// Mitsubishi GX Works2 project: PLC_Group_08   PLC: FX3G

// global labels: Global1
VAR_GLOBAL
  switch7 AT X007 : BOOL;
  lamp7 AT Y007 : BOOL;
  berry_input AT D1100 : INT;
  lemon_input AT D1102 : INT;
  stabilizer_input AT D1104 : INT;
  gum_input AT D1106 : INT;
  berry_stock AT D1200 : INT;
  lemon_stock AT D1202 : INT;
  stabilizer_stock AT D1204 : INT;
  gum_stock AT D1206 : INT;
  M_start AT M0 : BOOL;
  cooling_berry AT D1300 : INT;
  cooling_lemon AT D1302 : INT;
  storage AT D1304 : INT;
  switch5 AT X005 : BOOL;
  analog_input1 AT D8280 : INT;
  switch1 AT X001 : BOOL;
  save_analog_input1 AT D8202 : INT;
END_VAR
VAR_GLOBAL CONSTANT
  K_5 : INT := 2000;
  K_6 : INT := 2400;
  K_10 : INT := 4000;
END_VAR
VAR_GLOBAL
  M_normal AT M1 : BOOL;
  M_pinuk AT M2 : BOOL;
END_VAR
VAR_GLOBAL CONSTANT
  K_7 : INT := 7;
  K_berry_normal : INT := 280;
  K_berry_pinuk : INT := 385;
  K_lemon_normal : INT := 455;
  K_lemon_pinuk : INT := 665;
  K_gum_normal : INT := 28;
  K_gum_pinuk : INT := 70;
  K_stabilizer_normal : INT := 105;
  K_stabilizer_pinuk : INT := 210;
END_VAR
VAR_GLOBAL
  M_yes_stock AT M3 : BOOL;
  M_exit AT M4 : BOOL;
  berry_to_subtract AT D1500 : INT;
  lemon_to_subtract AT D1502 : INT;
  stabilizer_to_subtract AT D1504 : INT;
  gum_to_subtract AT D1506 : INT;
  making_berry AT D1306 : INT;
  making_lemon AT D1308 : INT;
  M_check_stock AT M5 : BOOL;
  M_make_icecream AT M6 : BOOL;
END_VAR
VAR_GLOBAL CONSTANT
  K_berry_total_normal : INT := 350;
  K_berry_total_pinuk : INT := 560;
  K_lemon_total_normal : INT := 490;
  K_lemon_total_pinuk : INT := 700;
END_VAR
VAR_GLOBAL
  berry_total AT D1508 : INT;
  lemon_total AT D1510 : INT;
  making_icecream_timer_c AT TC0 : BOOL;
END_VAR
VAR_GLOBAL CONSTANT
  K_50 : INT := 50;
END_VAR
VAR_GLOBAL
  making_icecream_timer_s AT TS0 : BOOL;
  lamp0 AT Y000 : BOOL;
  M_empty AT M7 : BOOL;
  M_cool_icecream AT M8 : BOOL;
  switch2 AT X002 : BOOL;
  cooling_icecream_timer_c AT TC1 : BOOL;
  cooling_icecream_timer_s AT TS1 : BOOL;
END_VAR
VAR_GLOBAL CONSTANT
  K_80 : INT := 80;
END_VAR
VAR_GLOBAL
  lamp2 AT Y002 : BOOL;
  switch3 AT X003 : BOOL;
  M_mix_materials AT M9 : BOOL;
  M_make_icecream_timer AT M11 : BOOL;
  M_cool_icecream_timer AT M10 : BOOL;
  mixing_container AT D1310 : INT;
END_VAR
VAR_GLOBAL CONSTANT
  K_mixing_total_normal : INT := 868;
  K_mixing_total_pinuk : INT := 1330;
  K_3 : INT := 3;
END_VAR
VAR_GLOBAL
  mixing_total AT D1512 : INT;
  mixing_duration AT D1514 : INT;
  M_mix_materials_timer AT M12 : BOOL;
  mix_materials_timer_c AT TC2 : BOOL;
  mix_materials_timer_s AT TS2 : BOOL;
  M_lamps_helper AT M13 : BOOL;
  lamp_5_timer_c AT TC3 : BOOL;
  lamp_5_timer_s AT TS3 : BOOL;
  lamp5 AT Y005 : BOOL;
  lamp_6_timer_c AT TC4 : BOOL;
  lamp_6_timer_s AT TS4 : BOOL;
  lamp6 AT Y006 : BOOL;
END_VAR
VAR_GLOBAL CONSTANT
  K_30 : INT := 30;
  K_01 : INT := 40;
  K_0 : INT;
END_VAR
VAR_GLOBAL
  M_berry_stock_check AT M14 : BOOL;
  M_lemon_stock_check AT M15 : BOOL;
  M_stabilizer_stock_check AT M16 : BOOL;
  M_gum_stock_check AT M17 : BOOL;
  analog_output AT D8282 : INT;
END_VAR
VAR_GLOBAL CONSTANT
  K_10_timer : INT := 10;
END_VAR
VAR_GLOBAL
  M_cool_and_mix AT M18 : BOOL;
END_VAR

// task Task_01 (event TRUE, interval 0, priority 31): POU_01

PROGRAM POU_01
(* structured ladder/FBD written out as ST: instructions are called as NAME(EN, inputs, outputs); _pN, _eN, _tN stand for wires *)
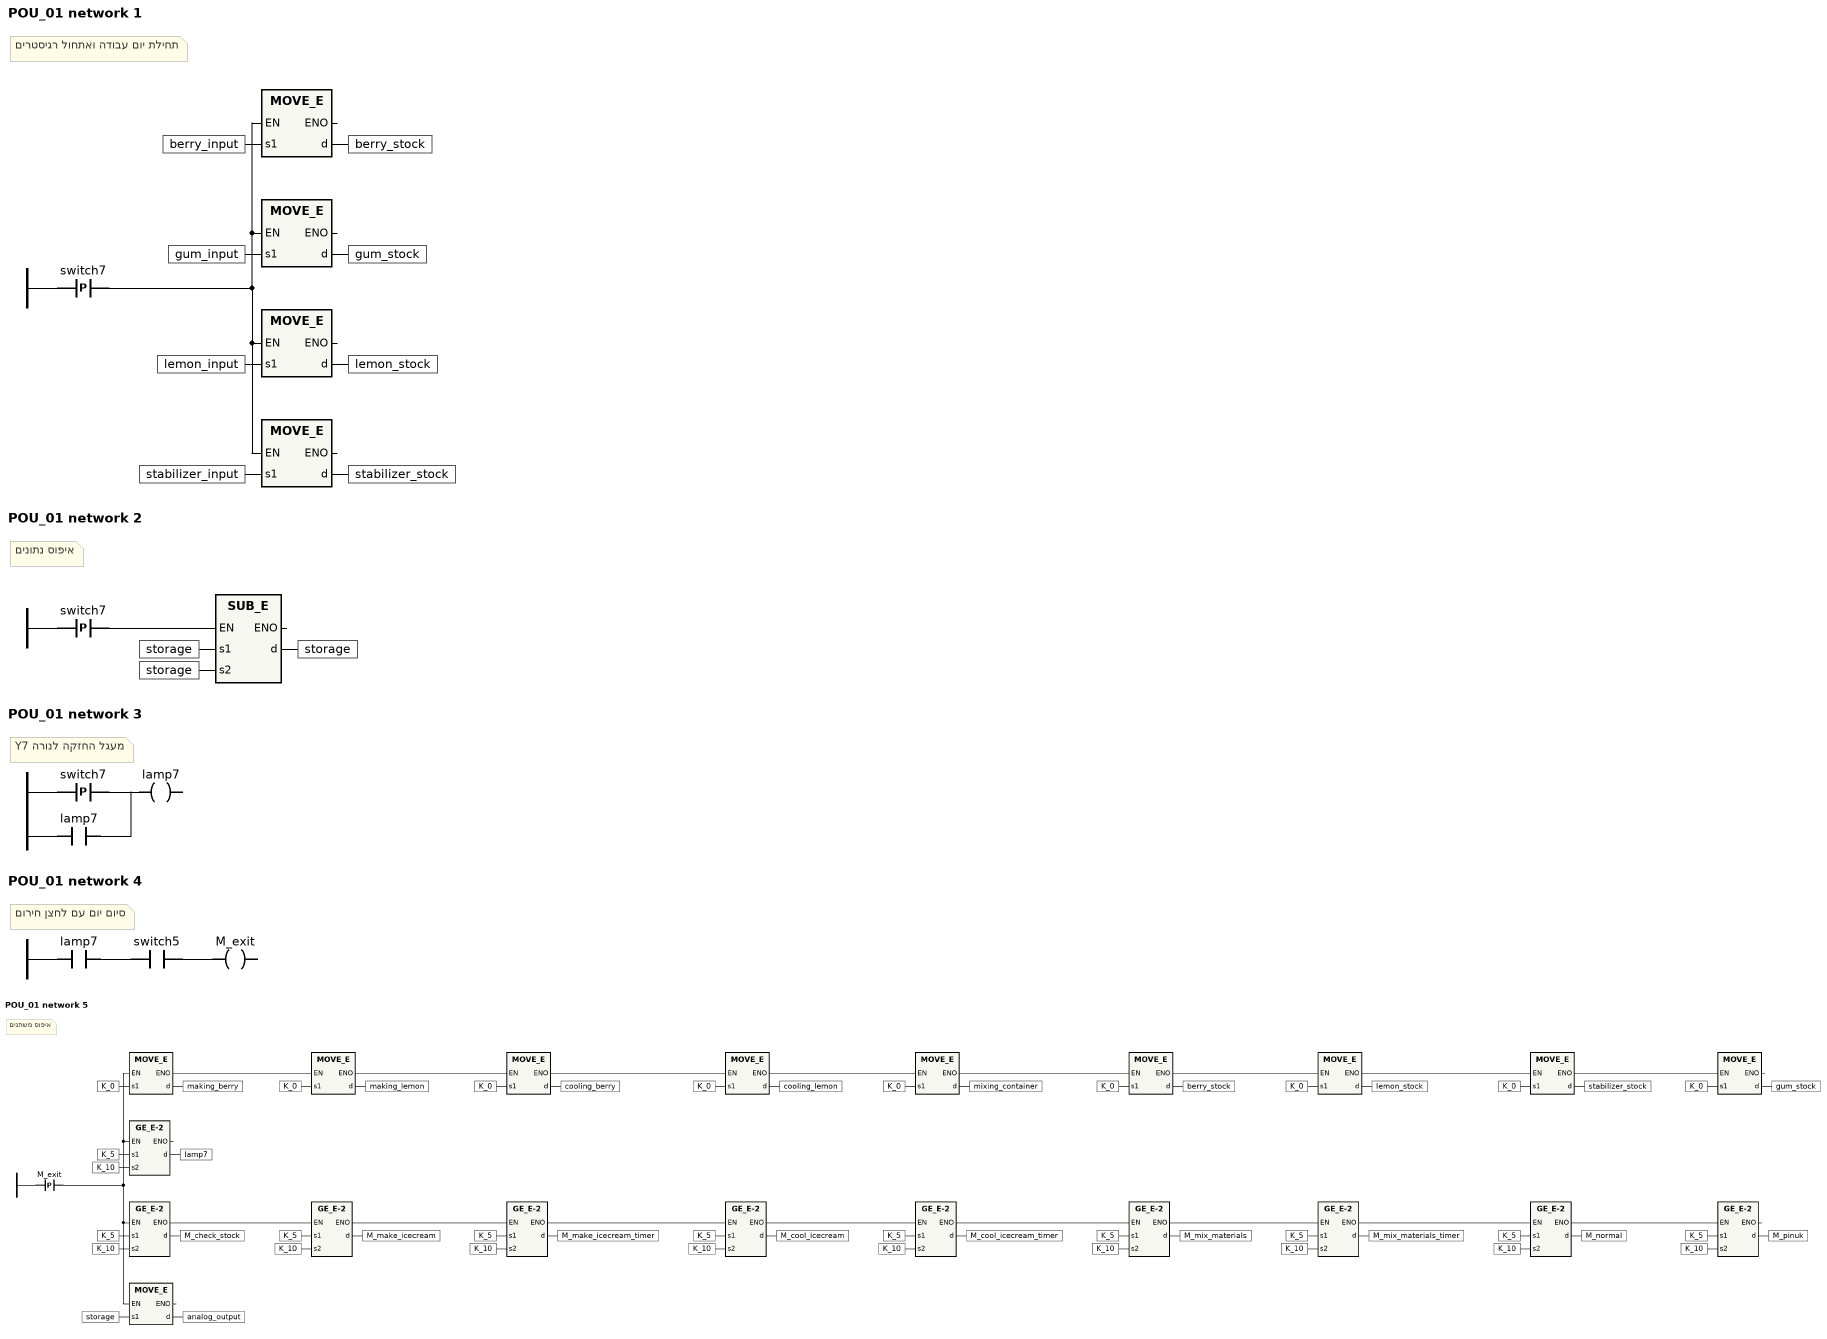
(* network 1 *)
(* תחילת יום עבודה ואתחול רגיסטרים *)
_p1 := LDP(TRUE, switch7);
MOVE_E(_p1, berry_input, berry_stock);
MOVE_E(_p1, gum_input, gum_stock);
MOVE_E(_p1, lemon_input, lemon_stock);
MOVE_E(_p1, stabilizer_input, stabilizer_stock);
(* network 2 *)
(* איפוס נתונים *)
SUB_E(LDP(TRUE, switch7), storage, storage, storage);
(* network 3 *)
(* מעגל החזקה לנורה Y7 *)
lamp7 := LDP(TRUE, switch7) OR lamp7;
(* network 4 *)
(* סיום יום עם לחצן חירום *)
M_exit := lamp7 AND switch5;
(* network 5 *)
(* איפוס משתנים *)
_p1 := LDP(TRUE, M_exit);
_e2 := MOVE_E(_p1, K_0, making_berry);
_e3 := MOVE_E(_e2, K_0, making_lemon);
_e4 := MOVE_E(_e3, K_0, cooling_berry);
_e5 := MOVE_E(_e4, K_0, cooling_lemon);
_e6 := MOVE_E(_e5, K_0, mixing_container);
_e7 := MOVE_E(_e6, K_0, berry_stock);
_e8 := MOVE_E(_e7, K_0, lemon_stock);
_e9 := MOVE_E(_e8, K_0, stabilizer_stock);
MOVE_E(_e9, K_0, gum_stock);
GE_E(_p1, K_5, K_10, lamp7);
_e10 := GE_E(_p1, K_5, K_10, M_check_stock);
_e11 := GE_E(_e10, K_5, K_10, M_make_icecream);
_e12 := GE_E(_e11, K_5, K_10, M_make_icecream_timer);
_e13 := GE_E(_e12, K_5, K_10, M_cool_icecream);
_e14 := GE_E(_e13, K_5, K_10, M_cool_icecream_timer);
_e15 := GE_E(_e14, K_5, K_10, M_mix_materials);
_e16 := GE_E(_e15, K_5, K_10, M_mix_materials_timer);
_e17 := GE_E(_e16, K_5, K_10, M_normal);
GE_E(_e17, K_5, K_10, M_pinuk);
MOVE_E(_p1, storage, analog_output);
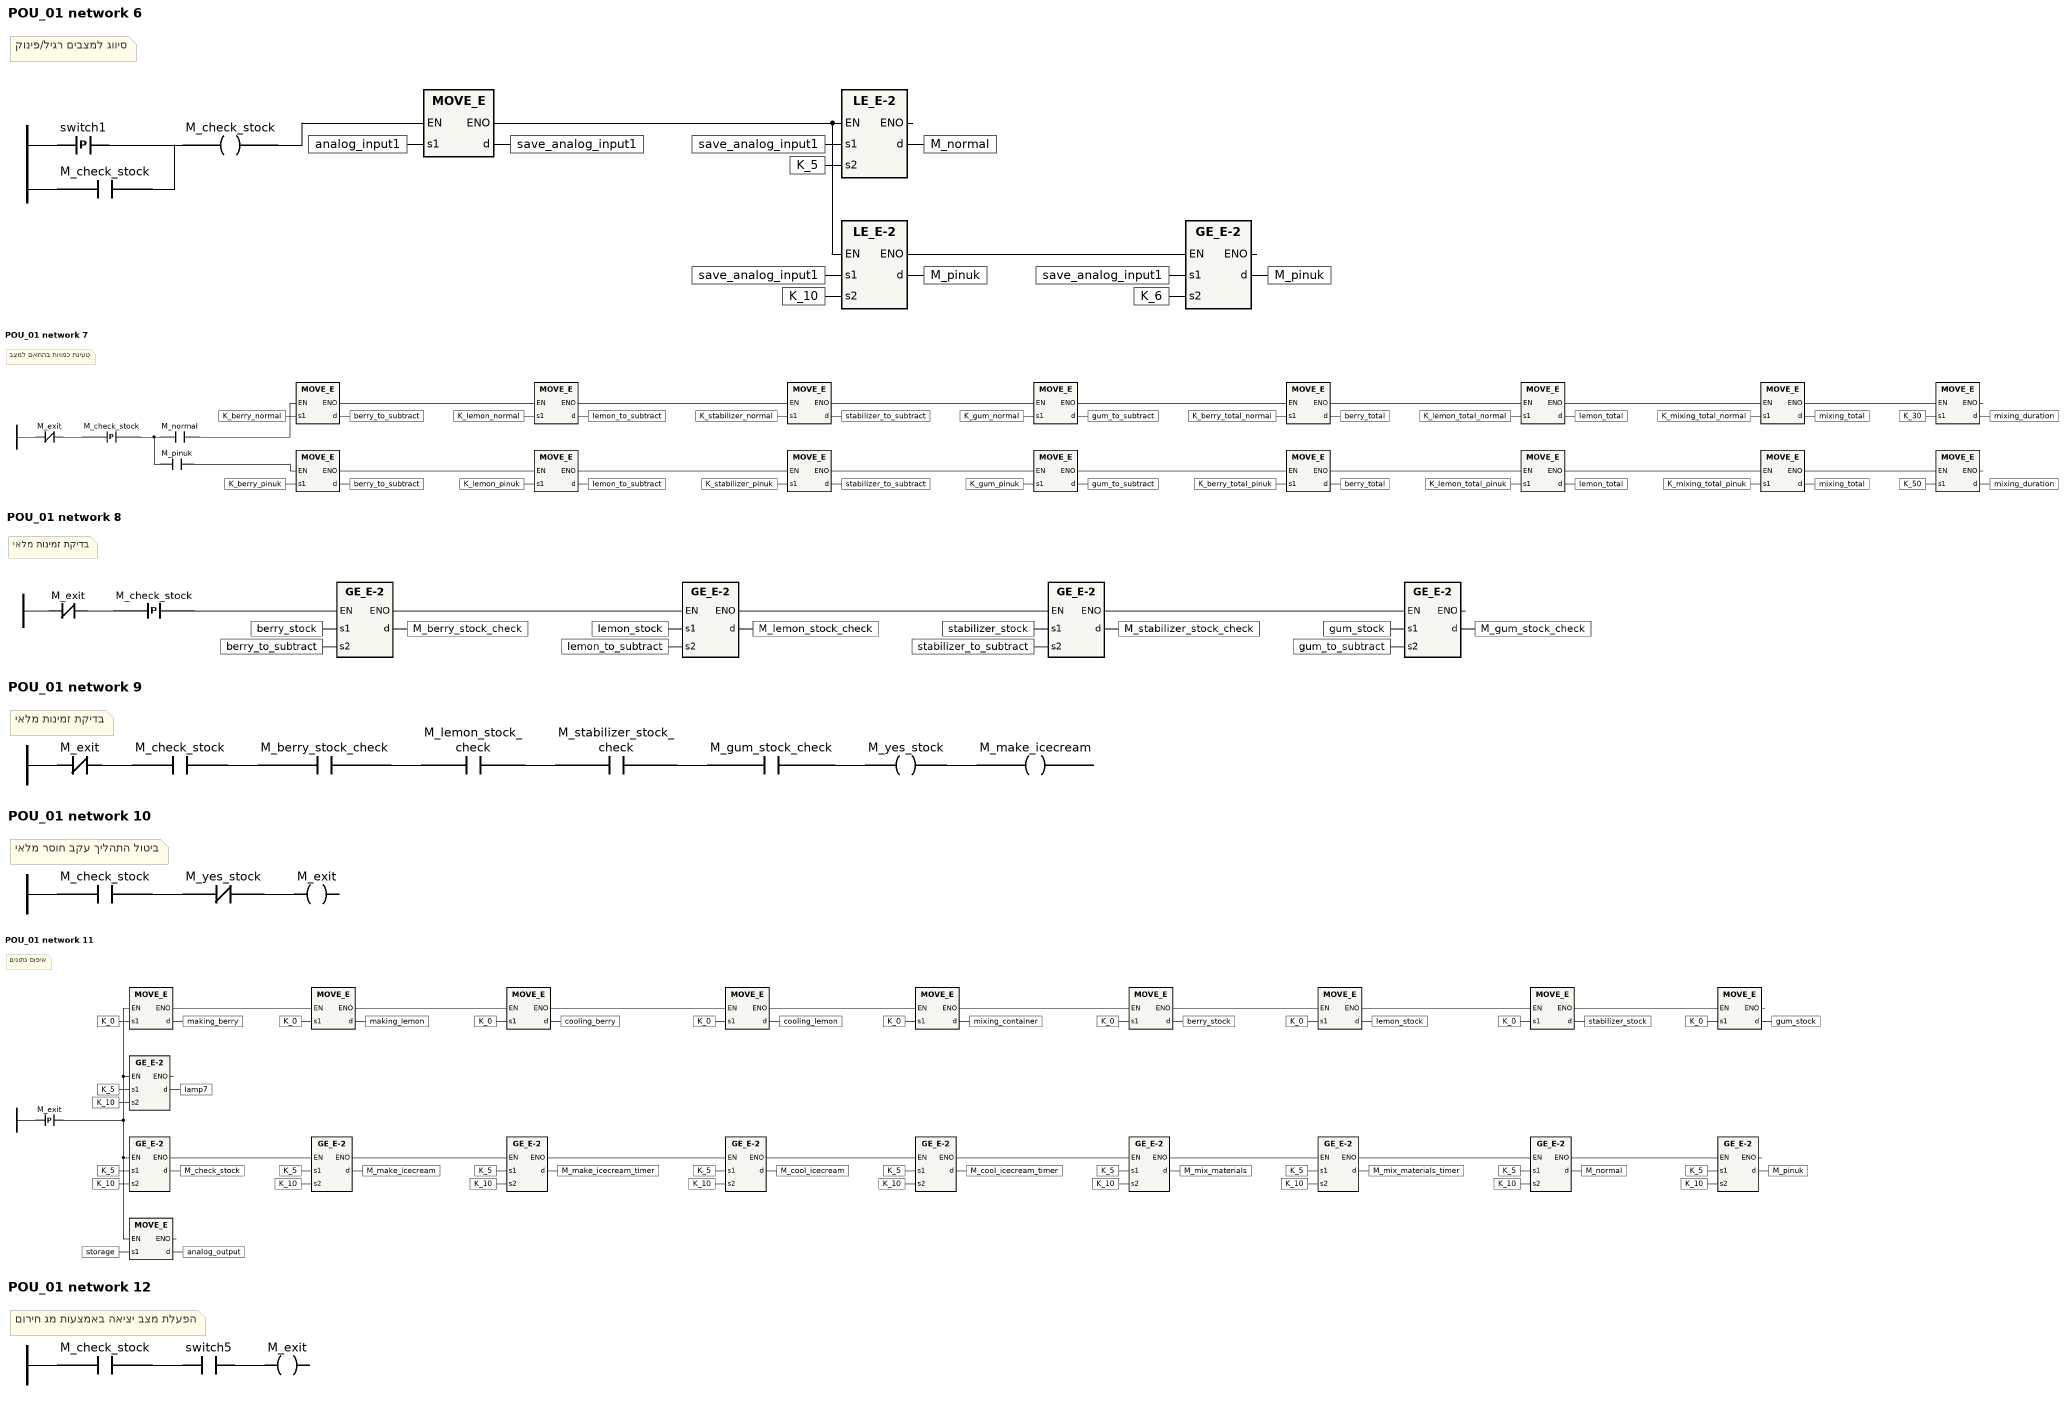
(* network 6 *)
(* סיווג למצבים רגיל/פינוק *)
_p1 := LDP(TRUE, switch1) OR M_check_stock;
M_check_stock := _p1;
_e2 := MOVE_E(_p1, analog_input1, save_analog_input1);
LE_E(_e2, save_analog_input1, K_5, M_normal);
_e3 := LE_E(_e2, save_analog_input1, K_10, M_pinuk);
GE_E(_e3, save_analog_input1, K_6, M_pinuk);
(* network 7 *)
(* טעינת כמויות בהתאם למצב *)
_p1 := NOT M_exit AND LDP(TRUE, M_check_stock);
_e2 := MOVE_E(_p1 AND M_normal, K_berry_normal, berry_to_subtract);
_e3 := MOVE_E(_e2, K_lemon_normal, lemon_to_subtract);
_e4 := MOVE_E(_e3, K_stabilizer_normal, stabilizer_to_subtract);
_e5 := MOVE_E(_e4, K_gum_normal, gum_to_subtract);
_e6 := MOVE_E(_e5, K_berry_total_normal, berry_total);
_e7 := MOVE_E(_e6, K_lemon_total_normal, lemon_total);
_e8 := MOVE_E(_e7, K_mixing_total_normal, mixing_total);
MOVE_E(_e8, K_30, mixing_duration);
_e9 := MOVE_E(_p1 AND M_pinuk, K_berry_pinuk, berry_to_subtract);
_e10 := MOVE_E(_e9, K_lemon_pinuk, lemon_to_subtract);
_e11 := MOVE_E(_e10, K_stabilizer_pinuk, stabilizer_to_subtract);
_e12 := MOVE_E(_e11, K_gum_pinuk, gum_to_subtract);
_e13 := MOVE_E(_e12, K_berry_total_pinuk, berry_total);
_e14 := MOVE_E(_e13, K_lemon_total_pinuk, lemon_total);
_e15 := MOVE_E(_e14, K_mixing_total_pinuk, mixing_total);
MOVE_E(_e15, K_50, mixing_duration);
(* network 8 *)
(* בדיקת זמינות מלאי *)
_e1 := GE_E(NOT M_exit AND LDP(TRUE, M_check_stock), berry_stock, berry_to_subtract, M_berry_stock_check);
_e2 := GE_E(_e1, lemon_stock, lemon_to_subtract, M_lemon_stock_check);
_e3 := GE_E(_e2, stabilizer_stock, stabilizer_to_subtract, M_stabilizer_stock_check);
GE_E(_e3, gum_stock, gum_to_subtract, M_gum_stock_check);
(* network 9 *)
(* בדיקת זמינות מלאי *)
_p1 := NOT M_exit AND M_check_stock AND M_berry_stock_check AND M_lemon_stock_check AND M_stabilizer_stock_check AND M_gum_stock_check;
M_yes_stock := _p1;
M_make_icecream := _p1;
(* network 10 *)
(* ביטול התהליך עקב חוסר מלאי *)
M_exit := M_check_stock AND NOT M_yes_stock;
(* network 11 *)
(* איפוס נתונים *)
_p1 := LDP(TRUE, M_exit);
_e2 := MOVE_E(_p1, K_0, making_berry);
_e3 := MOVE_E(_e2, K_0, making_lemon);
_e4 := MOVE_E(_e3, K_0, cooling_berry);
_e5 := MOVE_E(_e4, K_0, cooling_lemon);
_e6 := MOVE_E(_e5, K_0, mixing_container);
_e7 := MOVE_E(_e6, K_0, berry_stock);
_e8 := MOVE_E(_e7, K_0, lemon_stock);
_e9 := MOVE_E(_e8, K_0, stabilizer_stock);
MOVE_E(_e9, K_0, gum_stock);
GE_E(_p1, K_5, K_10, lamp7);
_e10 := GE_E(_p1, K_5, K_10, M_check_stock);
_e11 := GE_E(_e10, K_5, K_10, M_make_icecream);
_e12 := GE_E(_e11, K_5, K_10, M_make_icecream_timer);
_e13 := GE_E(_e12, K_5, K_10, M_cool_icecream);
_e14 := GE_E(_e13, K_5, K_10, M_cool_icecream_timer);
_e15 := GE_E(_e14, K_5, K_10, M_mix_materials);
_e16 := GE_E(_e15, K_5, K_10, M_mix_materials_timer);
_e17 := GE_E(_e16, K_5, K_10, M_normal);
GE_E(_e17, K_5, K_10, M_pinuk);
MOVE_E(_p1, storage, analog_output);
(* network 12 *)
(* הפעלת מצב יציאה באמצעות מג חירום *)
M_exit := M_check_stock AND switch5;
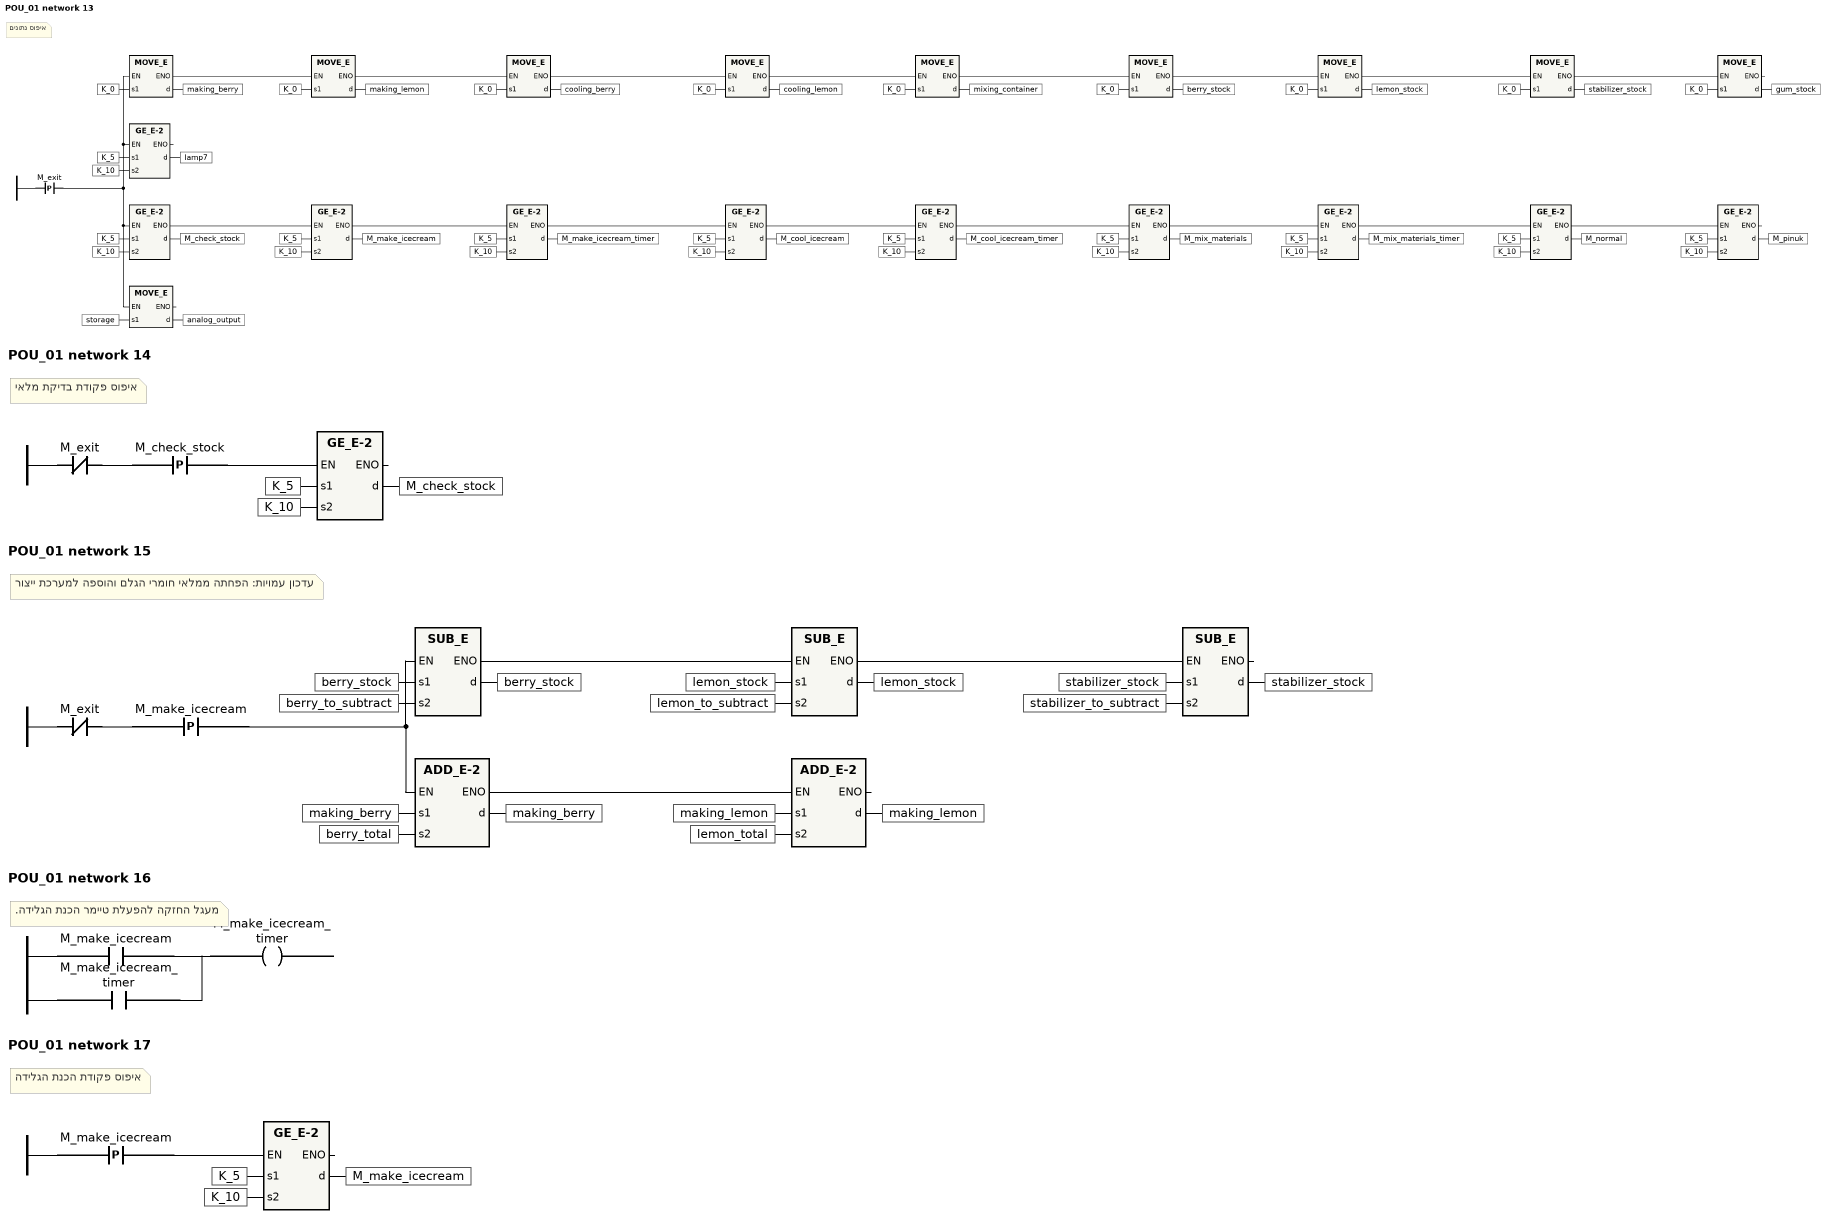
(* network 13 *)
(* איפוס נתונים *)
_p1 := LDP(TRUE, M_exit);
_e2 := MOVE_E(_p1, K_0, making_berry);
_e3 := MOVE_E(_e2, K_0, making_lemon);
_e4 := MOVE_E(_e3, K_0, cooling_berry);
_e5 := MOVE_E(_e4, K_0, cooling_lemon);
_e6 := MOVE_E(_e5, K_0, mixing_container);
_e7 := MOVE_E(_e6, K_0, berry_stock);
_e8 := MOVE_E(_e7, K_0, lemon_stock);
_e9 := MOVE_E(_e8, K_0, stabilizer_stock);
MOVE_E(_e9, K_0, gum_stock);
GE_E(_p1, K_5, K_10, lamp7);
_e10 := GE_E(_p1, K_5, K_10, M_check_stock);
_e11 := GE_E(_e10, K_5, K_10, M_make_icecream);
_e12 := GE_E(_e11, K_5, K_10, M_make_icecream_timer);
_e13 := GE_E(_e12, K_5, K_10, M_cool_icecream);
_e14 := GE_E(_e13, K_5, K_10, M_cool_icecream_timer);
_e15 := GE_E(_e14, K_5, K_10, M_mix_materials);
_e16 := GE_E(_e15, K_5, K_10, M_mix_materials_timer);
_e17 := GE_E(_e16, K_5, K_10, M_normal);
GE_E(_e17, K_5, K_10, M_pinuk);
MOVE_E(_p1, storage, analog_output);
(* network 14 *)
(* איפוס פקודת בדיקת מלאי *)
GE_E(NOT M_exit AND LDP(TRUE, M_check_stock), K_5, K_10, M_check_stock);
(* network 15 *)
(* עדכון עמויות: הפחתה ממלאי חומרי הגלם והוספה למערכת ייצור *)
_p1 := NOT M_exit AND LDP(TRUE, M_make_icecream);
_e2 := SUB_E(_p1, berry_stock, berry_to_subtract, berry_stock);
_e3 := SUB_E(_e2, lemon_stock, lemon_to_subtract, lemon_stock);
SUB_E(_e3, stabilizer_stock, stabilizer_to_subtract, stabilizer_stock);
_e4 := ADD_E(_p1, making_berry, berry_total, making_berry);
ADD_E(_e4, making_lemon, lemon_total, making_lemon);
(* network 16 *)
(* מעגל החזקה להפעלת טיימר הכנת הגלידה. *)
M_make_icecream_timer := M_make_icecream OR M_make_icecream_timer;
(* network 17 *)
(* איפוס פקודת הכנת הגלידה *)
GE_E(LDP(TRUE, M_make_icecream), K_5, K_10, M_make_icecream);
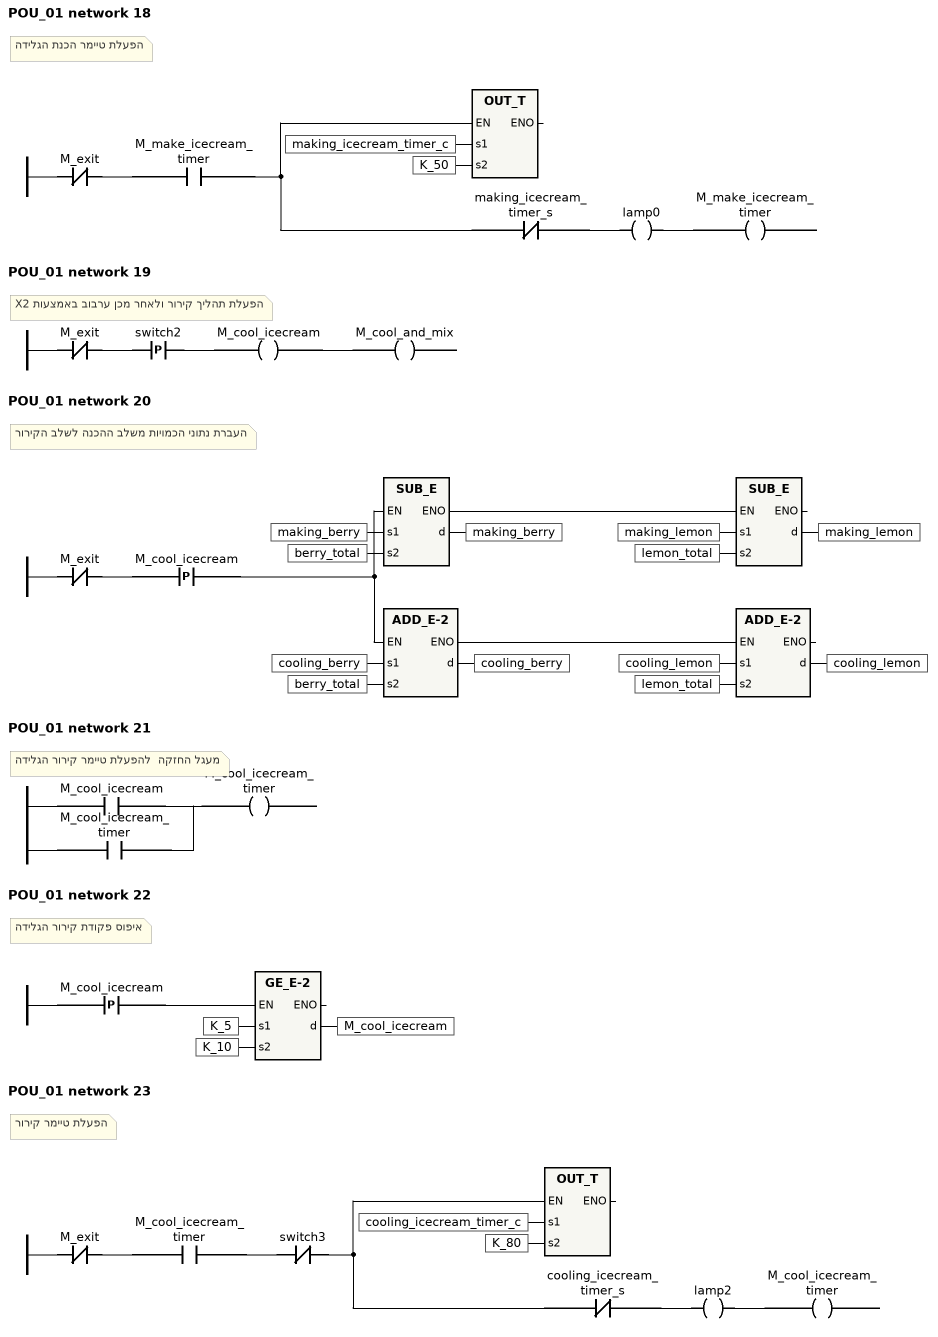
(* network 18 *)
(* הפעלת טיימר הכנת הגלידה *)
_p1 := NOT M_exit AND M_make_icecream_timer;
OUT_T(_p1, making_icecream_timer_c, K_50);
_p2 := _p1 AND NOT making_icecream_timer_s;
lamp0 := _p2;
M_make_icecream_timer := _p2;
(* network 19 *)
(* הפעלת תהליך קירור ולאחר מכן ערבוב באמצעות X2 *)
_p1 := NOT M_exit AND LDP(TRUE, switch2);
M_cool_icecream := _p1;
M_cool_and_mix := _p1;
(* network 20 *)
(* העברת נתוני הכמויות משלב ההכנה לשלב הקירור *)
_p1 := NOT M_exit AND LDP(TRUE, M_cool_icecream);
_e2 := SUB_E(_p1, making_berry, berry_total, making_berry);
SUB_E(_e2, making_lemon, lemon_total, making_lemon);
_e3 := ADD_E(_p1, cooling_berry, berry_total, cooling_berry);
ADD_E(_e3, cooling_lemon, lemon_total, cooling_lemon);
(* network 21 *)
(* מעגל החזקה  להפעלת טיימר קירור הגלידה *)
M_cool_icecream_timer := M_cool_icecream OR M_cool_icecream_timer;
(* network 22 *)
(* איפוס פקודת קירור הגלידה *)
GE_E(LDP(TRUE, M_cool_icecream), K_5, K_10, M_cool_icecream);
(* network 23 *)
(* הפעלת טיימר קירור *)
_p1 := NOT M_exit AND M_cool_icecream_timer AND NOT switch3;
OUT_T(_p1, cooling_icecream_timer_c, K_80);
_p2 := _p1 AND NOT cooling_icecream_timer_s;
lamp2 := _p2;
M_cool_icecream_timer := _p2;
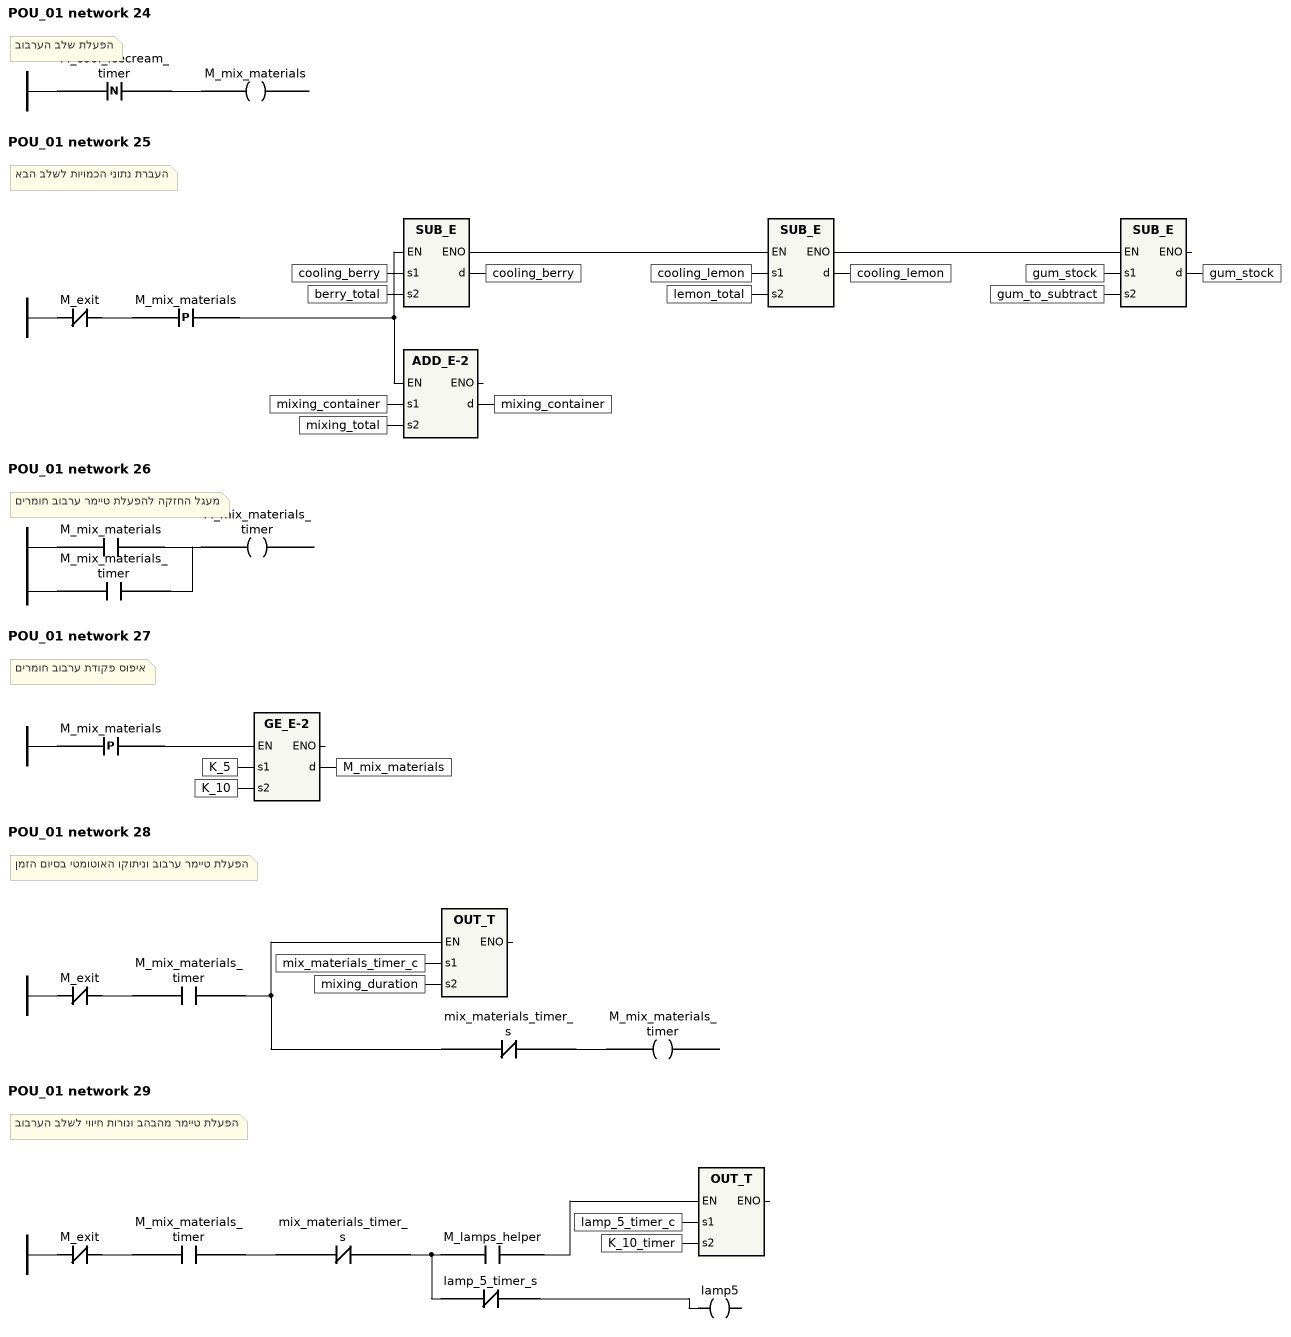
(* network 24 *)
(* הפעלת שלב הערבוב *)
M_mix_materials := LDF(TRUE, M_cool_icecream_timer);
(* network 25 *)
(* העברת נתוני הכמויות לשלב הבא *)
_p1 := NOT M_exit AND LDP(TRUE, M_mix_materials);
_e2 := SUB_E(_p1, cooling_berry, berry_total, cooling_berry);
_e3 := SUB_E(_e2, cooling_lemon, lemon_total, cooling_lemon);
SUB_E(_e3, gum_stock, gum_to_subtract, gum_stock);
ADD_E(_p1, mixing_container, mixing_total, mixing_container);
(* network 26 *)
(* מעגל החזקה להפעלת טיימר ערבוב חומרים *)
M_mix_materials_timer := M_mix_materials OR M_mix_materials_timer;
(* network 27 *)
(* איפוס פקודת ערבוב חומרים *)
GE_E(LDP(TRUE, M_mix_materials), K_5, K_10, M_mix_materials);
(* network 28 *)
(* הפעלת טיימר ערבוב וניתוקו האוטומטי בסיום הזמן *)
_p1 := NOT M_exit AND M_mix_materials_timer;
OUT_T(_p1, mix_materials_timer_c, mixing_duration);
M_mix_materials_timer := _p1 AND NOT mix_materials_timer_s;
(* network 29 *)
(* הפעלת טיימר מהבהב ונורות חיווי לשלב הערבוב *)
_p1 := NOT M_exit AND M_mix_materials_timer AND NOT mix_materials_timer_s;
OUT_T(_p1 AND M_lamps_helper, lamp_5_timer_c, K_10_timer);
lamp5 := _p1 AND NOT lamp_5_timer_s;
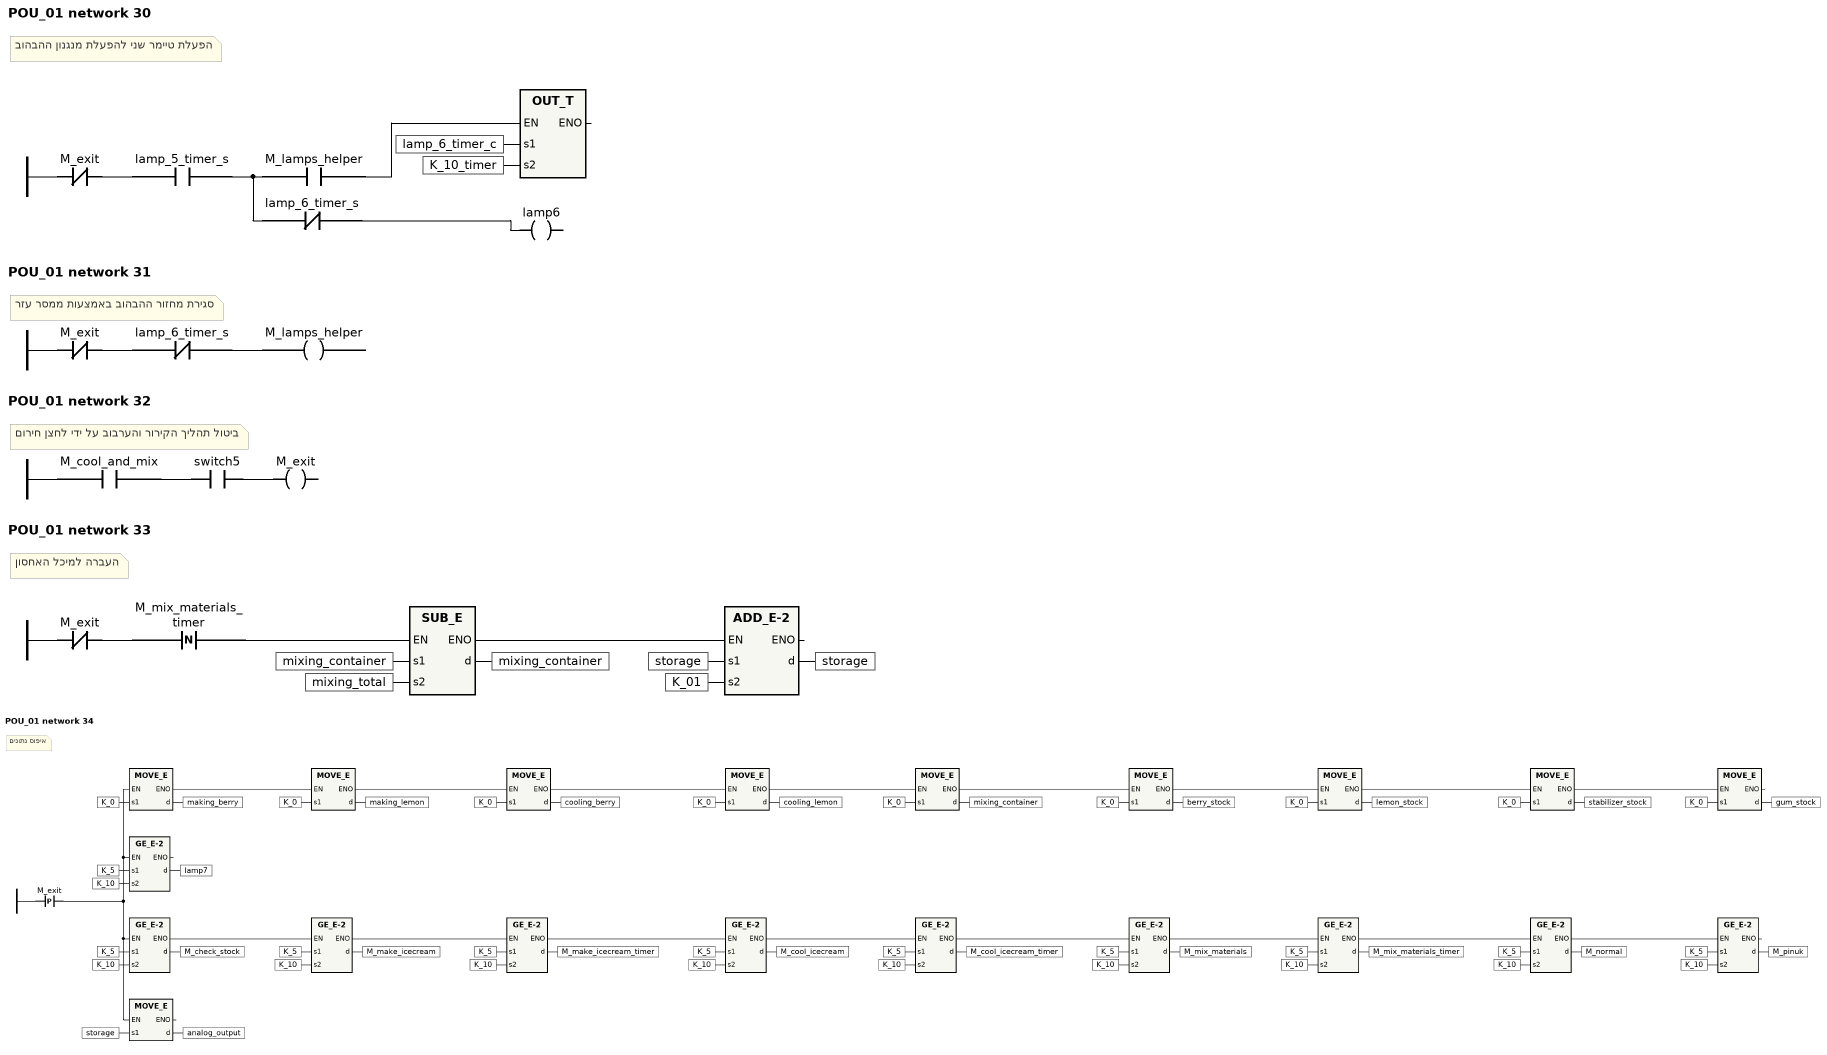
(* network 30 *)
(* הפעלת טיימר שני להפעלת מנגנון ההבהוב *)
_p1 := NOT M_exit AND lamp_5_timer_s;
OUT_T(_p1 AND M_lamps_helper, lamp_6_timer_c, K_10_timer);
lamp6 := _p1 AND NOT lamp_6_timer_s;
(* network 31 *)
(* סגירת מחזור ההבהוב באמצעות ממסר עזר *)
M_lamps_helper := NOT M_exit AND NOT lamp_6_timer_s;
(* network 32 *)
(* ביטול תהליך הקירור והערבוב על ידי לחצן חירום *)
M_exit := M_cool_and_mix AND switch5;
(* network 33 *)
(* העברה למיכל האחסון *)
_e1 := SUB_E(NOT M_exit AND LDF(TRUE, M_mix_materials_timer), mixing_container, mixing_total, mixing_container);
ADD_E(_e1, storage, K_01, storage);
(* network 34 *)
(* איפוס נתונים *)
_p1 := LDP(TRUE, M_exit);
_e2 := MOVE_E(_p1, K_0, making_berry);
_e3 := MOVE_E(_e2, K_0, making_lemon);
_e4 := MOVE_E(_e3, K_0, cooling_berry);
_e5 := MOVE_E(_e4, K_0, cooling_lemon);
_e6 := MOVE_E(_e5, K_0, mixing_container);
_e7 := MOVE_E(_e6, K_0, berry_stock);
_e8 := MOVE_E(_e7, K_0, lemon_stock);
_e9 := MOVE_E(_e8, K_0, stabilizer_stock);
MOVE_E(_e9, K_0, gum_stock);
GE_E(_p1, K_5, K_10, lamp7);
_e10 := GE_E(_p1, K_5, K_10, M_check_stock);
_e11 := GE_E(_e10, K_5, K_10, M_make_icecream);
_e12 := GE_E(_e11, K_5, K_10, M_make_icecream_timer);
_e13 := GE_E(_e12, K_5, K_10, M_cool_icecream);
_e14 := GE_E(_e13, K_5, K_10, M_cool_icecream_timer);
_e15 := GE_E(_e14, K_5, K_10, M_mix_materials);
_e16 := GE_E(_e15, K_5, K_10, M_mix_materials_timer);
_e17 := GE_E(_e16, K_5, K_10, M_normal);
GE_E(_e17, K_5, K_10, M_pinuk);
MOVE_E(_p1, storage, analog_output);
END_PROGRAM
